// TIA Portal V21 export
FUNCTION_BLOCK "LineAnimationFb"   // FB802, LAD
{ S7_Optimized_Access := 'FALSE' }
// stored: AutoNumber false, SetENOAutomatically false
   VAR_INPUT
      AlwaysTrue : Bool;
      AlwaysFalse : Bool;
      SecPulse : Bool;
      "Spare 1" : Bool;
      "Spare 2" : Bool;
      "Spare 3" : Bool;
      "Spare 4" : Bool;
      "Spare 5" : Bool;
   END_VAR
   VAR_OUTPUT
      LineColour : DInt;
      ValveColour : DInt;
      ColourTemp : Int;
      Mode : Int;   // 0 - Force Close, 1- AutoOn, 2-ForceOn
      SpareOp2 : Int;
      Output : Bool;
      AutoOn : Bool;
      AutoOff : Bool;
      ManualOn : Bool;
      ManualOpen : Bool;
      ManualClose : Bool;
      V01 { ExternalAccessible := 'False'; ExternalVisible := 'False'; ExternalWritable := 'False'} : "LineAnimation";
      V02 { ExternalAccessible := 'False'; ExternalVisible := 'False'; ExternalWritable := 'False'} : "LineAnimation";
      V03 { ExternalAccessible := 'False'; ExternalVisible := 'False'; ExternalWritable := 'False'} : "LineAnimation";
      V04 { ExternalAccessible := 'False'; ExternalVisible := 'False'; ExternalWritable := 'False'} : "LineAnimation";
      V05 { ExternalAccessible := 'False'; ExternalVisible := 'False'; ExternalWritable := 'False'} : "LineAnimation";
      V06 { ExternalAccessible := 'False'; ExternalVisible := 'False'; ExternalWritable := 'False'} : "LineAnimation";
      V07 { ExternalAccessible := 'False'; ExternalVisible := 'False'; ExternalWritable := 'False'} : "LineAnimation";
      V08 { ExternalAccessible := 'False'; ExternalVisible := 'False'; ExternalWritable := 'False'} : "LineAnimation";
      V09 { ExternalAccessible := 'False'; ExternalVisible := 'False'; ExternalWritable := 'False'} : "LineAnimation";
      V10 { ExternalAccessible := 'False'; ExternalVisible := 'False'; ExternalWritable := 'False'} : "LineAnimation";
      V11 { ExternalAccessible := 'False'; ExternalVisible := 'False'; ExternalWritable := 'False'} : "LineAnimation";
      V12 { ExternalAccessible := 'False'; ExternalVisible := 'False'; ExternalWritable := 'False'} : "LineAnimation";
      V13 { ExternalAccessible := 'False'; ExternalVisible := 'False'; ExternalWritable := 'False'} : "LineAnimation";
      V14 { ExternalAccessible := 'False'; ExternalVisible := 'False'; ExternalWritable := 'False'} : "LineAnimation";
      V15 { ExternalAccessible := 'False'; ExternalVisible := 'False'; ExternalWritable := 'False'} : "LineAnimation";
      V16 { ExternalAccessible := 'False'; ExternalVisible := 'False'; ExternalWritable := 'False'} : "LineAnimation";
      V17 { ExternalAccessible := 'False'; ExternalVisible := 'False'; ExternalWritable := 'False'} : "LineAnimation";
      V18 { ExternalAccessible := 'False'; ExternalVisible := 'False'; ExternalWritable := 'False'} : "LineAnimation";
      V19 { ExternalAccessible := 'False'; ExternalVisible := 'False'; ExternalWritable := 'False'} : "LineAnimation";
      V20 { ExternalAccessible := 'False'; ExternalVisible := 'False'; ExternalWritable := 'False'} : "LineAnimation";
   END_VAR
BEGIN

REGION Network 1: Auto On
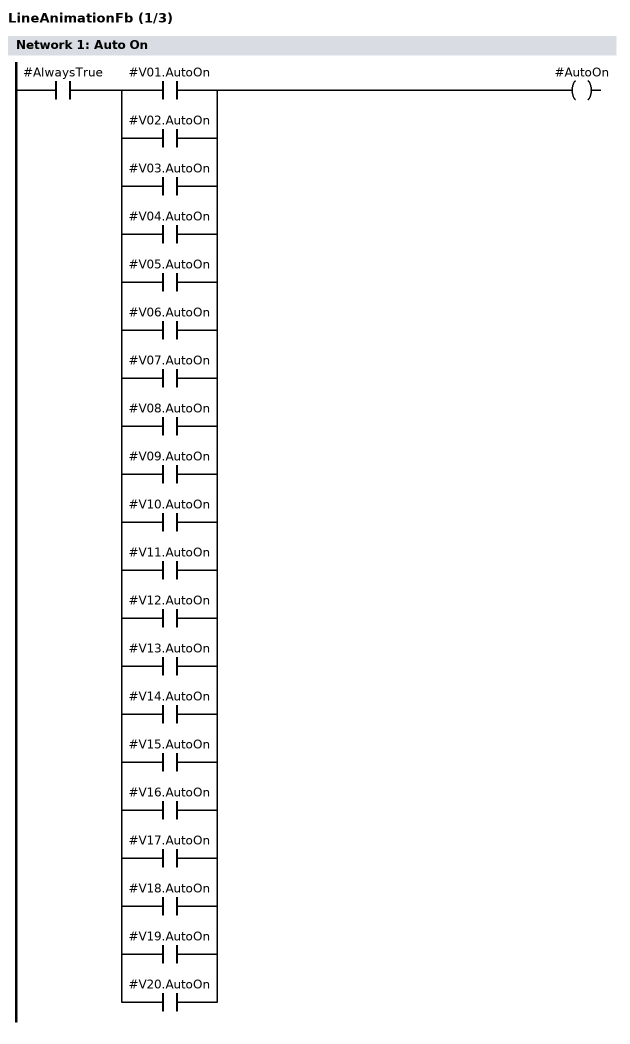
   RUNG wire#powerrail
      Contact( #AlwaysTrue )
      wire#w1
      Contact( #V01.AutoOn )
      wire#w2
      Coil( #AutoOn )
   END_RUNG
   RUNG wire#w1
      Contact( #V02.AutoOn )
   END_RUNG wire#w2
   RUNG wire#w1
      Contact( #V03.AutoOn )
   END_RUNG wire#w2
   RUNG wire#w1
      Contact( #V04.AutoOn )
   END_RUNG wire#w2
   RUNG wire#w1
      Contact( #V05.AutoOn )
   END_RUNG wire#w2
   RUNG wire#w1
      Contact( #V06.AutoOn )
   END_RUNG wire#w2
   RUNG wire#w1
      Contact( #V07.AutoOn )
   END_RUNG wire#w2
   RUNG wire#w1
      Contact( #V08.AutoOn )
   END_RUNG wire#w2
   RUNG wire#w1
      Contact( #V09.AutoOn )
   END_RUNG wire#w2
   RUNG wire#w1
      Contact( #V10.AutoOn )
   END_RUNG wire#w2
   RUNG wire#w1
      Contact( #V11.AutoOn )
   END_RUNG wire#w2
   RUNG wire#w1
      Contact( #V12.AutoOn )
   END_RUNG wire#w2
   RUNG wire#w1
      Contact( #V13.AutoOn )
   END_RUNG wire#w2
   RUNG wire#w1
      Contact( #V14.AutoOn )
   END_RUNG wire#w2
   RUNG wire#w1
      Contact( #V15.AutoOn )
   END_RUNG wire#w2
   RUNG wire#w1
      Contact( #V16.AutoOn )
   END_RUNG wire#w2
   RUNG wire#w1
      Contact( #V17.AutoOn )
   END_RUNG wire#w2
   RUNG wire#w1
      Contact( #V18.AutoOn )
   END_RUNG wire#w2
   RUNG wire#w1
      Contact( #V19.AutoOn )
   END_RUNG wire#w2
   RUNG wire#w1
      Contact( #V20.AutoOn )
   END_RUNG wire#w2
   // the same network as SCL:
   #AutoOn := #AlwaysTrue AND (#V01.AutoOn OR #V02.AutoOn OR #V03.AutoOn OR #V04.AutoOn OR #V05.AutoOn OR #V06.AutoOn OR #V07.AutoOn OR #V08.AutoOn OR #V09.AutoOn OR #V10.AutoOn OR #V11.AutoOn OR #V12.AutoOn OR #V13.AutoOn OR #V14.AutoOn OR #V15.AutoOn OR #V16.AutoOn OR #V17.AutoOn OR #V18.AutoOn OR #V19.AutoOn OR #V20.AutoOn);
END_REGION

REGION Network 2: Force Open
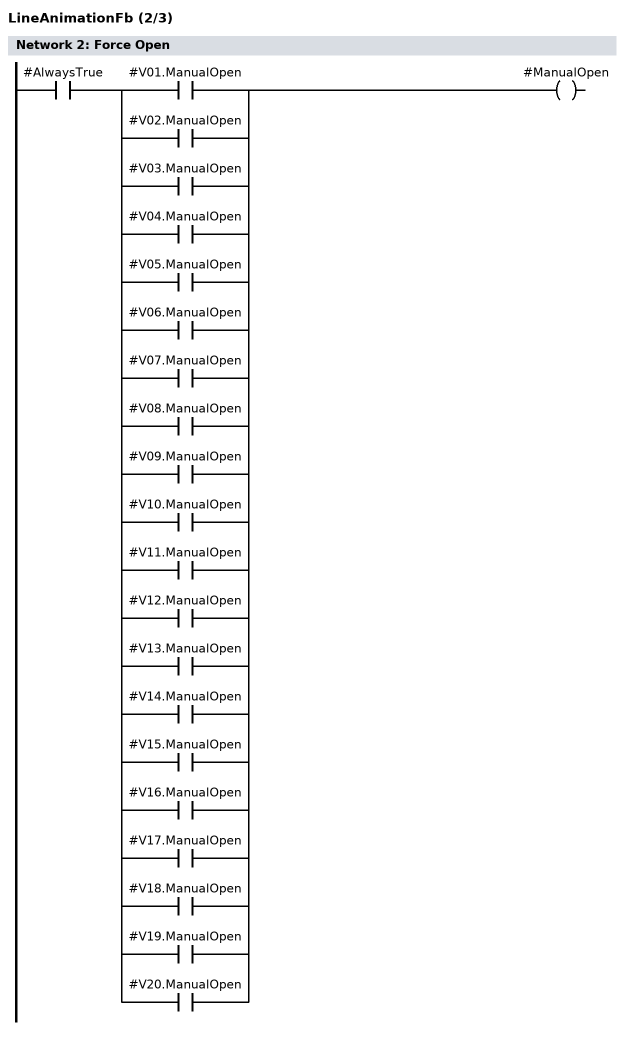
   RUNG wire#powerrail
      Contact( #AlwaysTrue )
      wire#w1
      Contact( #V01.ManualOpen )
      wire#w2
      Coil( #ManualOpen )
   END_RUNG
   RUNG wire#w1
      Contact( #V02.ManualOpen )
   END_RUNG wire#w2
   RUNG wire#w1
      Contact( #V03.ManualOpen )
   END_RUNG wire#w2
   RUNG wire#w1
      Contact( #V04.ManualOpen )
   END_RUNG wire#w2
   RUNG wire#w1
      Contact( #V05.ManualOpen )
   END_RUNG wire#w2
   RUNG wire#w1
      Contact( #V06.ManualOpen )
   END_RUNG wire#w2
   RUNG wire#w1
      Contact( #V07.ManualOpen )
   END_RUNG wire#w2
   RUNG wire#w1
      Contact( #V08.ManualOpen )
   END_RUNG wire#w2
   RUNG wire#w1
      Contact( #V09.ManualOpen )
   END_RUNG wire#w2
   RUNG wire#w1
      Contact( #V10.ManualOpen )
   END_RUNG wire#w2
   RUNG wire#w1
      Contact( #V11.ManualOpen )
   END_RUNG wire#w2
   RUNG wire#w1
      Contact( #V12.ManualOpen )
   END_RUNG wire#w2
   RUNG wire#w1
      Contact( #V13.ManualOpen )
   END_RUNG wire#w2
   RUNG wire#w1
      Contact( #V14.ManualOpen )
   END_RUNG wire#w2
   RUNG wire#w1
      Contact( #V15.ManualOpen )
   END_RUNG wire#w2
   RUNG wire#w1
      Contact( #V16.ManualOpen )
   END_RUNG wire#w2
   RUNG wire#w1
      Contact( #V17.ManualOpen )
   END_RUNG wire#w2
   RUNG wire#w1
      Contact( #V18.ManualOpen )
   END_RUNG wire#w2
   RUNG wire#w1
      Contact( #V19.ManualOpen )
   END_RUNG wire#w2
   RUNG wire#w1
      Contact( #V20.ManualOpen )
   END_RUNG wire#w2
   // the same network as SCL:
   #ManualOpen := #AlwaysTrue AND (#V01.ManualOpen OR #V02.ManualOpen OR #V03.ManualOpen OR #V04.ManualOpen OR #V05.ManualOpen OR #V06.ManualOpen OR #V07.ManualOpen OR #V08.ManualOpen OR #V09.ManualOpen OR #V10.ManualOpen OR #V11.ManualOpen OR #V12.ManualOpen OR #V13.ManualOpen OR #V14.ManualOpen OR #V15.ManualOpen OR #V16.ManualOpen OR #V17.ManualOpen OR #V18.ManualOpen OR #V19.ManualOpen OR #V20.ManualOpen);
END_REGION

REGION Network 3: Line Colour
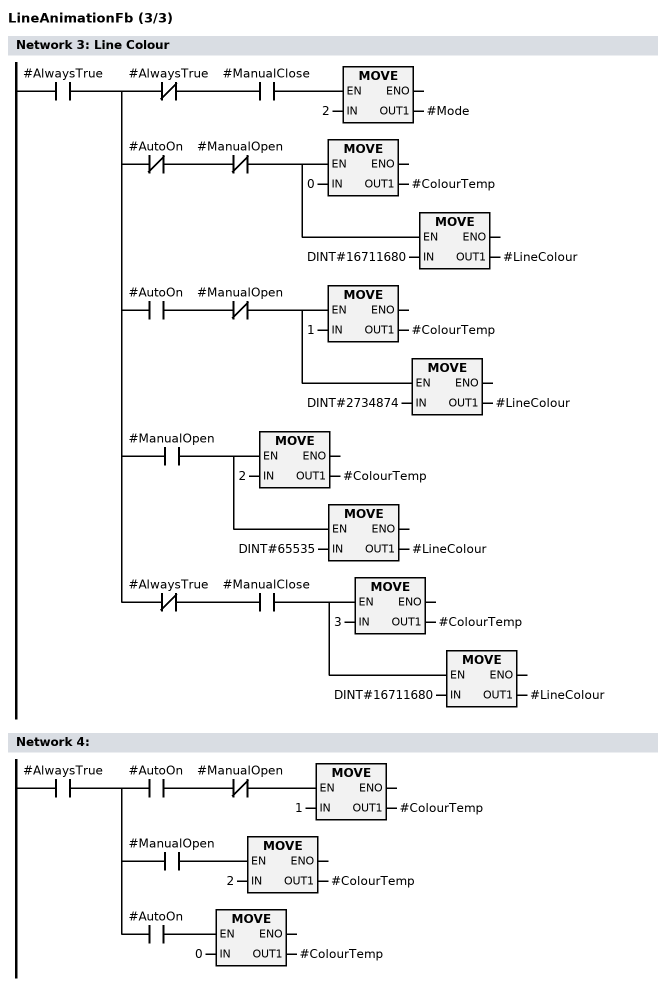
   RUNG wire#powerrail
      Contact( #AlwaysTrue )
      wire#w1
      I_Contact( #AlwaysTrue )
      Contact( #ManualClose )
      Move(in := 2, out1 => #Mode)
   END_RUNG
   RUNG wire#w1
      I_Contact( #AutoOn )
      I_Contact( #ManualOpen )
      wire#w2
      Move(in := 0, out1 => #ColourTemp)
   END_RUNG
   RUNG wire#w2
      Move(in := DINT#16711680, out1 => #LineColour)
   END_RUNG
   RUNG wire#w1
      Contact( #AutoOn )
      I_Contact( #ManualOpen )
      wire#w3
      Move(in := 1, out1 => #ColourTemp)
   END_RUNG
   RUNG wire#w3
      Move(in := DINT#2734874, out1 => #LineColour)
   END_RUNG
   RUNG wire#w1
      Contact( #ManualOpen )
      wire#w4
      Move(in := 2, out1 => #ColourTemp)
   END_RUNG
   RUNG wire#w4
      Move(in := DINT#65535, out1 => #LineColour)
   END_RUNG
   RUNG wire#w1
      I_Contact( #AlwaysTrue )
      Contact( #ManualClose )
      wire#w5
      Move(in := 3, out1 => #ColourTemp)
   END_RUNG
   RUNG wire#w5
      Move(in := DINT#16711680, out1 => #LineColour)
   END_RUNG
   // the same network as SCL:
   IF #AlwaysTrue AND NOT #AlwaysTrue AND #ManualClose THEN #Mode := 2; END_IF;
   IF #AlwaysTrue AND NOT #AutoOn AND NOT #ManualOpen THEN
       #ColourTemp := 0;
       #LineColour := DINT#16711680;
   END_IF;
   IF #AlwaysTrue AND #AutoOn AND NOT #ManualOpen THEN
       #ColourTemp := 1;
       #LineColour := DINT#2734874;
   END_IF;
   IF #AlwaysTrue AND #ManualOpen THEN
       #ColourTemp := 2;
       #LineColour := DINT#65535;
   END_IF;
   IF #AlwaysTrue AND NOT #AlwaysTrue AND #ManualClose THEN
       #ColourTemp := 3;
       #LineColour := DINT#16711680;
   END_IF;
END_REGION

REGION Network 4
   RUNG wire#powerrail
      Contact( #AlwaysTrue )
      wire#w1
      Contact( #AutoOn )
      I_Contact( #ManualOpen )
      Move(in := 1, out1 => #ColourTemp)
   END_RUNG
   RUNG wire#w1
      Contact( #ManualOpen )
      Move(in := 2, out1 => #ColourTemp)
   END_RUNG
   RUNG wire#w1
      Contact( #AutoOn )
      Move(in := 0, out1 => #ColourTemp)
   END_RUNG
   // the same network as SCL:
   IF #AlwaysTrue AND #AutoOn AND NOT #ManualOpen THEN #ColourTemp := 1; END_IF;
   IF #AlwaysTrue AND #ManualOpen THEN #ColourTemp := 2; END_IF;
   IF #AlwaysTrue AND #AutoOn THEN #ColourTemp := 0; END_IF;
END_REGION
END_FUNCTION_BLOCK
